// TIA Portal V15.1 export
// export: Created 2026-01-15T16:29:46.0427253Z, ExportSetting WithDefaults, WithReadOnly, DisplayName Totally Integrated Automation Portal, DisplayVersion V15.1 Update 8, DisplayName TIA Portal Openness, DisplayVersion V15.1 Update 8, DisplayName STEP 7 Professional, DisplayVersion V15.1 Update 8, DisplayName WinCC Advanced, DisplayVersion V15.1 Update 8
DATA_BLOCK "C#4_WD_WEIGHT"   // DB4
{ S7_Optimized_Access := 'FALSE' }
VERSION : 0.1
// stored: AutoNumber true, CodeModifiedDate 2026-01-10T09:51:14.6601717Z, CompileDate 2026-01-15T16:25:51.96112Z, CreationDate 2026-01-15T16:23:32.6582836Z, DBAccessibleFromOPCUA true, InterfaceModifiedDate 2026-01-10T09:51:14.6601717Z, IsConsistent true, IsKnowHowProtected false, IsOnlyStoredInLoadMemory false, IsPLCDB false, IsWriteProtectedInAS false, ModifiedDate 2026-01-10T15:14:24.5843652Z, ParameterModified 2026-01-10T09:51:14.6601717Z, StructureModified 2026-01-10T09:51:14.6601717Z
   VAR RETAIN
      "W_AG1_TG.DLC" : Real;   // Phễu cân Cốt liệu 1_Thời gian trễ cân
      "W_AG1_TG.DLX" : Real;   // Phễu cân Cốt liệu 1_Thời gian trễ xả
      "W_AG1_TG.DLD" : Real;   // Phễu cân Cốt liệu 1_Thời gian trễ đóng cân
      "W_AG1_KL.BRO" : Real;   // Phễu cân Cốt liệu 1_Khối lượng báo rỗng
      "W_AG1_KL.RUG" : Real;   // Phễu cân Cốt liệu 1_Khối lượng rung cân
      "W_AG1_TG.ON_RUNG" : Real;   // Phễu cân Cốt liệu 1_Thời gian bật rung
      "W_AG1_TG.OF_RUNG" : Real;   // Phễu cân Cốt liệu 1_Thời gian tắt rung
      "W_FD1_TG.DLC" : Real;   // Phễu cân FD 1_Thời gian trễ cân
      "W_FD1_TG.DLX" : Real;   // Phễu cân FD 1_Thời gian trễ xả
      "W_FD1_TG.DLD" : Real;   // Phễu cân FD 1_Thời gian trễ đóng cân
      "W_FD1_KL.BRO" : Real;   // Phễu cân FD 1_Khối lượng báo rỗng
      "W_FD1_KL.RUG" : Real;   // Phễu cân FD1_Khối lượng rung cân
      "W_FD1_TG.ON_RUNG" : Real;   // Phễu cân FD 1_Thời gian bật rung
      "W_FD1_TG.OF_RUNG" : Real;   // Phễu cân FD 1_Thời gian tắt rung
      "W_AP1_TG.DLC" : Real;   // Phễu cân Nhựa 1_Thời gian trễ cân
      "W_AP1_TG.DLX" : Real;   // Phễu cân Nhựa 1_Thời gian trễ xả
      "W_AP1_TG.DLD" : Real;   // Phễu cân Nhựa 1_Thời gian trễ đóng cân
      "W_AP1_KL.BRO" : Real;   // Phễu cân Nhựa 1_Khối lượng báo rỗng
      "W_SB1_TG.DLC" : Real;   // Phễu cân SBS 1_Thời gian trễ cân
      "W_SB1_TG.DLX" : Real;   // Phễu cân SBS 1_Thời gian trễ xả
      "W_SB1_TG.DLD" { ExternalWritable := 'False'} : Real;   // Phễu cân SBS 1_Thời gian trễ đóng cân
      "W_SB1_KL.BRO" : Real;   // Phễu cân SBS 1_Khối lượng báo rỗng
      "W_SB1_KL.RUG" : Real;   // Phễu cân SBS 1_Khối lượng rung cân
      "W_SB1_TG.ON_RUNG" : Real;   // Phễu cân SBS 1_Thời gian bật rung
      "W_SB1_TG.OF_RUNG" : Real;   // Phễu cân SBS 1_Thời gian tắt rung
      SO_ME_TRON : Real;   // Số mẻ cần trộn
      SV_AG1 : Real;   // Khối lượng Cần cân Cốt liệu 1
      SV_AG2 : Real;   // Khối lượng Cần cân Cốt liệu 2
      SV_AG3 : Real;   // Khối lượng Cần cân Cốt liệu 3
      SV_AG4 : Real;   // Khối lượng Cần cân Cốt liệu 4
      SV_AG5 : Real;   // Khối lượng Cần cân Cốt liệu 5
      SV_FD1 : Real;   // Khối lượng Cần cân FD 1
      SV_AP1 : Real;   // Khối lượng Cần cân Nhựa 1
      SV_SB1 : Real;   // Khối lượng Cần cân SBS 1
      "W_IND_AGG1_TG.DLC" : Real;   // Phễu cân IND Cốt liệu 1_Thời gian trễ cân
      "W_IND_AGG1_TG.DLX" : Real;   // Phễu cân IND Cốt liệu 1_Thời gian trễ xả
      "W_IND_AGG1_TG.DLD" : Real;   // Phễu cân IND Cốt liệu 1_Thời gian trễ đóng cân
      "W_IND_AGG1_KL.BRO" : Real;   // Phễu cân IND Cốt liệu 1_Khối lượng báo rỗng
      "W_IND_AGG1_KL.RUG" : Real;   // Phễu cân IND Cốt liệu 1_Khối lượng rung cân
      "W_IND_AGG1_TG.ON_RUNG" : Real;   // Phễu cân IND Cốt liệu 1_Thời gian bật rung
      "W_IND_AGG1_TG.OF_RUNG" : Real;   // Phễu cân IND Cốt liệu 1_Thời gian tắt rung
      "W_IND_AGG2_TG.DLC" : Real;   // Phễu cân IND Cốt liệu 2_Thời gian trễ cân
      "W_IND_AGG2_TG.DLX" : Real;   // Phễu cân IND Cốt liệu 2_Thời gian trễ xả
      "W_IND_AGG2_TG.DLD" : Real;   // Phễu cân IND Cốt liệu 2_Thời gian trễ đóng cân
      "W_IND_AGG2_KL.BRO" : Real;   // Phễu cân IND Cốt liệu 2_Khối lượng báo rỗng
      "W_IND_AGG2_KL.RUG" : Real;   // Phễu cân IND Cốt liệu 2_Khối lượng rung cân
      "W_IND_AGG2_TG.ON_RUNG" : Real;   // Phễu cân IND Cốt liệu 2_Thời gian bật rung
      "W_IND_AGG2_TG.OF_RUNG" : Real;   // Phễu cân IND Cốt liệu 2_Thời gian tắt rung
      "W_IND_AGG3_TG.DLC" : Real;   // Phễu cân IND Cốt liệu 3_Thời gian trễ cân
      "W_IND_AGG3_TG.DLX" : Real;   // Phễu cân IND Cốt liệu 3_Thời gian trễ xả
      "W_IND_AGG3_TG.DLD" : Real;   // Phễu cân IND Cốt liệu 3_Thời gian trễ đóng cân
      "W_IND_AGG3_KL.BRO" : Real;   // Phễu cân IND Cốt liệu 3_Khối lượng báo rỗng
      "W_IND_AGG3_KL.RUG" : Real;   // Phễu cân IND Cốt liệu 3_Khối lượng rung cân
      "W_IND_AGG3_TG.ON_RUNG" : Real;   // Phễu cân IND Cốt liệu 3_Thời gian bật rung
      "W_IND_AGG3_TG.OF_RUNG" : Real;   // Phễu cân IND Cốt liệu 3_Thời gian tắt rung
      "W_IND_AGG4_TG.DLC" : Real;   // Phễu cân IND Cốt liệu 4_Thời gian trễ cân
      "W_IND_AGG4_TG.DLX" : Real;   // Phễu cân IND Cốt liệu 4_Thời gian trễ xả
      "W_IND_AGG4_TG.DLD" : Real;   // Phễu cân IND Cốt liệu 4_Thời gian trễ đóng cân
      "W_IND_AGG4_KL.BRO" : Real;   // Phễu cân IND Cốt liệu 4_Khối lượng báo rỗng
      "W_IND_AGG4_KL.RUG" : Real;   // Phễu cân IND Cốt liệu 4_Khối lượng rung cân
      "W_IND_AGG4_TG.ON_RUNG" : Real;   // Phễu cân IND Cốt liệu 4_Thời gian bật rung
      "W_IND_AGG4_TG.OF_RUNG" : Real;   // Phễu cân IND Cốt liệu 4_Thời gian tắt rung
      "W_IND_AGG5_TG.DLC" : Real;   // Phễu cân IND Cốt liệu 5_Thời gian trễ cân
      "W_IND_AGG5_TG.DLX" : Real;   // Phễu cân IND Cốt liệu 5_Thời gian trễ xả
      "W_IND_AGG5_TG.DLD" : Real;   // Phễu cân IND Cốt liệu 5_Thời gian trễ đóng cân
      "W_IND_AGG5_KL.BRO" : Real;   // Phễu cân IND Cốt liệu 5_Khối lượng báo rỗng
      "W_IND_AGG5_KL.RUG" : Real;   // Phễu cân IND Cốt liệu 5_Khối lượng rung cân
      "W_IND_AGG5_TG.ON_RUNG" : Real;   // Phễu cân IND Cốt liệu 5_Thời gian bật rung
      "W_IND_AGG5_TG.OF_RUNG" : Real;   // Phễu cân IND Cốt liệu 5_Thời gian tắt rung
   END_VAR
BEGIN
END_DATA_BLOCK
